VISUALIZATION VisuMMA  // 2x2
END_VISUALIZATION

(* stored: Version 1.1.0.1, ProductVersion 3.1.4020.12
   Visu VisuMMA: Id {22beceb3-43c5-47f8-a6b8-79a61dbbe16d} *)
